(* PLC project  *)

CONFIGURATION XF71
END_CONFIGURATION
